PROGRAM Input_Mapping
VAR
	
END_VAR

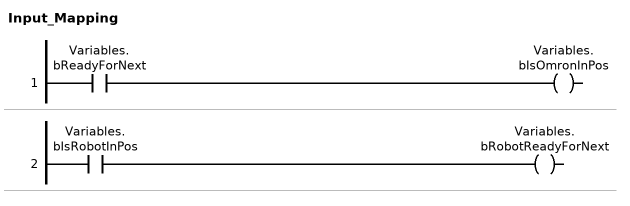
// NETWORK 1
Variables.bIsOmronInPos := Variables.bReadyForNext;

// NETWORK 2
Variables.bRobotReadyForNext := Variables.bIsRobotInPos;

END_PROGRAM

(* stored: Version 1.1.0.1, ProductVersion 3.1.4020.6
   POU Input_Mapping: Id {41e9298a-49db-4e65-9ff3-b01c7f6d6767}, SpecialFunc None *)
